TYPE ST_MachineControl_HMI :
STRUCT
	bAutomaticMode 		: BOOL;
	bServiceMode		: BOOL;
	
	bStartProcess		: BOOL;
	bPauseProcess		: BOOL;
	bStopProcess		: BOOL;
	
	
END_STRUCT
END_TYPE

(* stored: Version 1.1.0.1
   DUT ST_MachineControl_HMI: Id {37d31d4c-cf1e-460c-bd71-06e22e4ecc38} *)
